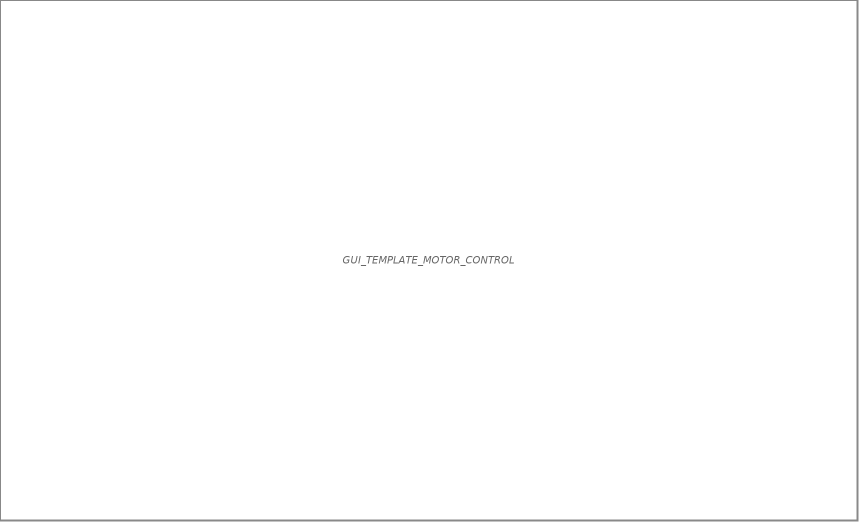
VISUALIZATION GUI_DROT_Motor  // 859x522
    Frame (0,0 857x520)
        shows GUI_TEMPLATE_MOTOR_CONTROL(m_Instance := MAIN.drot.motor)
END_VISUALIZATION

(* stored: Version 1.1.0.1, ProductVersion 3.1.4022.16
   Visu GUI_DROT_Motor: Id {10e2555f-3553-4341-b637-a4d664e73584} *)
